// TIA Portal V16 export
// export: Created 2023-10-30T22:43:51.2917106Z, ExportSetting WithDefaults, DisplayName Totally Integrated Automation Portal, DisplayVersion V16, DisplayName TIA Portal Version Control Interface, DisplayVersion V16, DisplayName TIA Portal Openness, DisplayVersion V16, DisplayName SINAMICS Startdrive Advanced, DisplayVersion V16, DisplayName SINAMICS Startdrive G130, G150, S120, S150, SINAMICS MV, S210, DisplayVersion V16, DisplayName SINAMICS Startdrive G110M, G120, G120C, G120D, G120P, DisplayVersion V16, DisplayName STEP 7 Professional, DisplayVersion V16, DisplayName STEP 7 Safety, DisplayVersion V16, DisplayName WinCC Professional, DisplayVersion V16
DATA_BLOCK "DataLogCreate_DB"   // DB12
// stored: AutoNumber true, DBAccessibleFromOPCUA true, InstanceOfName DataLogCreate_SFB, OfSystemLibElement DataLogCreate, OfSystemLibVersion 1.0
"DataLogCreate_SFB"
   // VAR_INPUT
   //    REQ : Bool;
   //    Records : UDInt;
   //    Format : UInt;
   //    Timestamp : UInt;
   //    "Name" : Variant;
   // END_VAR
   // VAR_OUTPUT
   //    DONE : Bool;
   //    BUSY : Bool;
   //    ERROR : Bool;
   //    STATUS : Word;
   // END_VAR
   // VAR_IN_OUT
   //    ID : DWord;
   //    Header : Variant;
   //    Data : Variant;
   // END_VAR
BEGIN
END_DATA_BLOCK
